// SIMATIC S7-200 project (STEP 7-Micro/WIN), CPU 222 REL 01.22

SYMBOL_TABLE USUARIO1
FR1              I0.0     // RELE TERMICO
S1               I0.1     // PULSADOR PARO
S2               I0.2     // PULSADOR MARCHA
KM1              Q0.0     // CONTACTOR LINEA
KM2              Q0.1     // CONTACTOR ESTRELLA
KM3              Q0.2     // CONTACTOR TRIANGULO
H1               Q0.3     // SEÑALIZACION MARCHA
H2               Q0.4     // SEÑALIACION AVERIA
H3               Q0.5     // SEÑALIZACION PARADA
END_SYMBOL_TABLE

ORGANIZATION_BLOCK PRINCIPAL:OB1
TITLE=COMENTARIOS DEL PROGRAMA
BEGIN
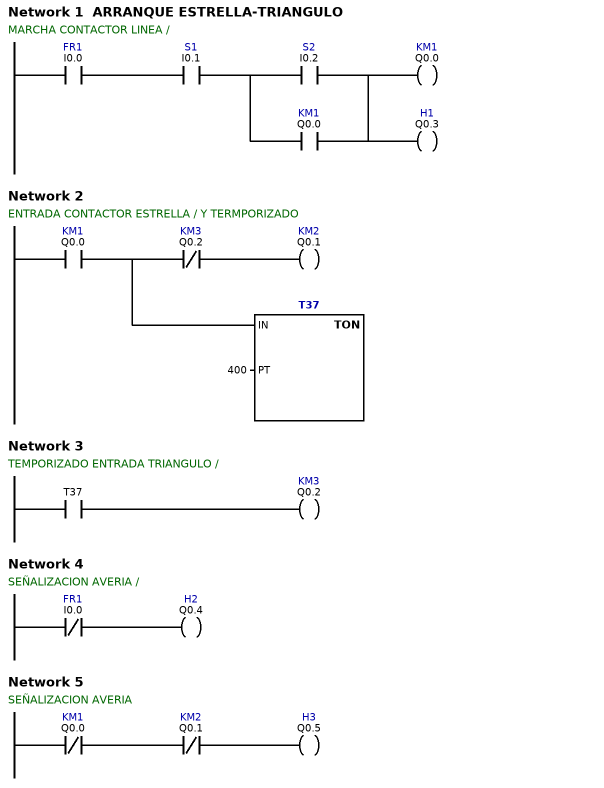
Network 1 // ARRANQUE ESTRELLA-TRIANGULO

// MARCHA CONTACTOR LINEA
// 
LD     FR1:I0.0
A      S1:I0.1
LD     S2:I0.2
O      KM1:Q0.0
ALD
=      KM1:Q0.0
=      H1:Q0.3
Network 2
// ENTRADA CONTACTOR ESTRELLA
// Y TERMPORIZADO
LD     KM1:Q0.0
LPS
AN     KM3:Q0.2
=      KM2:Q0.1
LPP
TON    T37, 400
Network 3
// TEMPORIZADO ENTRADA TRIANGULO
// 
// (network saved uncompiled; LAD cells follow)
// row 0: c0 -| |- T37  c1 --  c2 -( ) KM3:Q0.2
Network 4
// SEÑALIZACION AVERIA
// 
LDN    FR1:I0.0
=      H2:Q0.4
Network 5
// SEÑALIZACION AVERIA
LDN    KM1:Q0.0
AN     KM2:Q0.1
=      H3:Q0.5
END_ORGANIZATION_BLOCK
